(* IEC 61131-3 sources: julia_exos_development/src/exos_julia/exos_julia, 2 files *)

(* ---- exos_julia.typ ---- *)
TYPE
	IntStruct_typ : 	STRUCT
		MyInt13 : UDINT;
		MyInt14 : ARRAY[0..2]OF USINT;
		MyInt133 : UDINT;
		MyInt124 : ARRAY[0..2]OF USINT;
	END_STRUCT;
	IntStruct1_typ : 	STRUCT
		MyInt13 : UDINT;
	END_STRUCT;
	IntStruct2_typ : 	STRUCT
		MyInt23 : UDINT;
		MyInt24 : ARRAY[0..3]OF USINT;
		MyInt25 : UDINT;
	END_STRUCT;
	exos_julia : 	STRUCT
		MyInt1 : UDINT; (*PUB*)
		MyInt3 : ARRAY[0..4]OF USINT; (*PUB SUB*)
	END_STRUCT;
END_TYPE

(* ---- exos_julia.fun ---- *)
FUNCTION_BLOCK exos_juliaInit
	VAR_OUTPUT
		Handle : UDINT;
	END_VAR
	VAR
		_state : USINT;
	END_VAR
END_FUNCTION_BLOCK

FUNCTION_BLOCK exos_juliaCyclic
	VAR_INPUT
		Enable : BOOL;
		Handle : UDINT;
		Start : BOOL;
		pexos_julia : REFERENCE TO exos_julia;
	END_VAR
	VAR_OUTPUT
		Active : BOOL;
		Error : BOOL;
		Disconnected : BOOL;
		Connected : BOOL;
		Operational : BOOL;
		Aborted : BOOL;
	END_VAR
	VAR
		_state : USINT;
	END_VAR
END_FUNCTION_BLOCK

FUNCTION_BLOCK exos_juliaExit
	VAR_INPUT
		Handle : UDINT;
	END_VAR
	VAR
		_state : USINT;
	END_VAR
END_FUNCTION_BLOCK
